TYPE DigitalInputBase_50022E7B :
STRUCT
END_STRUCT
END_TYPE

(* stored: Version 1.2.0.0, ProductVersion 3.1.4024.9
   DUT DigitalInputBase_50022E7B: Id {9667b2fd-9461-45ab-9d38-a633ecc0e723} *)
